// TIA Portal V17 export
// export: Created 2023-02-13T11:16:49.8587223Z, ExportSetting WithDefaults, DisplayName Totally Integrated Automation Portal, DisplayVersion V17, DisplayName TIA Portal Openness, DisplayVersion V17, DisplayName TIA Portal Teamcenter Gateway, DisplayVersion V17, DisplayName TIA Portal Version Control Interface, DisplayVersion V17, DisplayName SINAMICS Startdrive Advanced, DisplayVersion V17, DisplayName SINAMICS Startdrive G130, G150, S120, S150, SINAMICS MV, S210, DisplayVersion V17, DisplayName SINAMICS Startdrive G110M, G120, G120C, G120D, G120P, G115D, DisplayVersion V17, DisplayName STEP 7 Professional, DisplayVersion V17, DisplayName STEP 7 Safety, DisplayVersion V17, DisplayName WinCC Professional, DisplayVersion V17
DATA_BLOCK "General Buffer"   // DB63
{ S7_Optimized_Access := 'TRUE' }
VERSION : 0.1
// stored: AutoNumber true, DBAccessibleFromOPCUA true, DBAccessibleFromWebserver true, IsOnlyStoredInLoadMemory false, IsRetainMemResEnabled false, IsWriteProtectedInAS false, MemoryReserve 100
   VAR
      "CIP Enable" : Struct
         Cluster1_Line3 : Bool;
         Cluster2_Line1 : Bool;
         Cluster2_Line2 : Bool;
         Cluster2_Line3 : Bool;
      END_STRUCT;
      "CIP Line Open" : Struct
         Cluster1_Line3 : Bool;
         Cluster2_Line1 : Bool;
         Cluster2_Line2 : Bool;
         Cluster2_Line3 : Bool;
      END_STRUCT;
   END_VAR
BEGIN
END_DATA_BLOCK
